{attribute 'GeneratedUsingTerminal: EL7201-0001-0017'}
{attribute addProperty BoxType "EL7201-0001-0017"}
{attribute addProperty Id "ControlwordAT %Q*UINT2"}
{attribute addProperty CRC "4092675873"}
{attribute addProperty Size "2"}
TYPE DS402_Controlword_F3F14721 :
STRUCT
	{attribute addProperty Name "Controlword"}
	Controlword AT %Q* : UINT;
END_STRUCT
END_TYPE

(* stored: Version 1.2.0.0, ProductVersion 3.1.4024.9
   DUT DS402_Controlword_F3F14721: Id {b5ce75bb-ec6e-4350-b3f0-f6275322acb4} *)
